// TIA Portal project "3M-9" (V16)

(* hardware
DEVICE "S7-1200 station_1"  S7-1200 Station
   slot 0: "Rack_0"  S7-1200 Rack  Rack  V1.0
   slot 1: "PLC_1"  CPU 1212C AC/DC/Rly  6ES7 212-1BE40-0XB0  V4.4
*)

// ===== PLC "PLC_1"  CPU 1212C AC/DC/Rly =====

VAR_GLOBAL   // PLC tag table "Default tag table"
   "START" AT %I0.0 : Bool;
   "STOP" AT %I0.1 : Bool;
   "MOTOR1" AT %Q0.0 : Bool;
   "MOTOR2" AT %Q0.1 : Bool;
   "MOTOR3" AT %Q0.2 : Bool;
   "X" AT %M0.0 : Bool;
   "Case 1" AT %M0.1 : Bool;
   "Case 2" AT %M0.2 : Bool;
   "Case 3" AT %M0.3 : Bool;
   "Y" AT %M0.4 : Bool;
   "tm1" AT %M0.5 : Bool;
   "tm2" AT %M0.6 : Bool;
   "TM3" AT %M0.7 : Bool;
   "SAVE Y" AT %M1.0 : Bool;
   "SAVE Z" AT %M1.1 : Bool;
END_VAR

// folder: System blocks/Program resources

DATA_BLOCK "timer1"   // DB1
{ S7_Optimized_Access := 'TRUE' }
AUTHOR : Simatic
FAMILY : IEC
NAME : IEC_TMR
VERSION : 1.0
// stored: InstanceOfName IEC_TIMER
"IEC_TIMER"
BEGIN
END_DATA_BLOCK

DATA_BLOCK "TIMER2"   // DB2
{ S7_Optimized_Access := 'TRUE' }
AUTHOR : Simatic
FAMILY : IEC
NAME : IEC_TMR
VERSION : 1.0
// stored: InstanceOfName IEC_TIMER
"IEC_TIMER"
BEGIN
END_DATA_BLOCK

DATA_BLOCK "TIMER3"   // DB3
{ S7_Optimized_Access := 'TRUE' }
AUTHOR : Simatic
FAMILY : IEC
NAME : IEC_TMR
VERSION : 1.0
// stored: InstanceOfName IEC_TIMER
"IEC_TIMER"
BEGIN
END_DATA_BLOCK

// folder: (top level)

ORGANIZATION_BLOCK "Main"   // OB1, LAD, ProgramCycle
TITLE = "Main Program Sweep (Cycle)"
{ S7_Optimized_Access := 'TRUE' }
VERSION : 0.1
   VAR_INPUT
      Initial_Call : Bool;   // Initial call of this OB
      Remanence : Bool;   // =True, if remanent data are available
   END_VAR
BEGIN

REGION Network 1
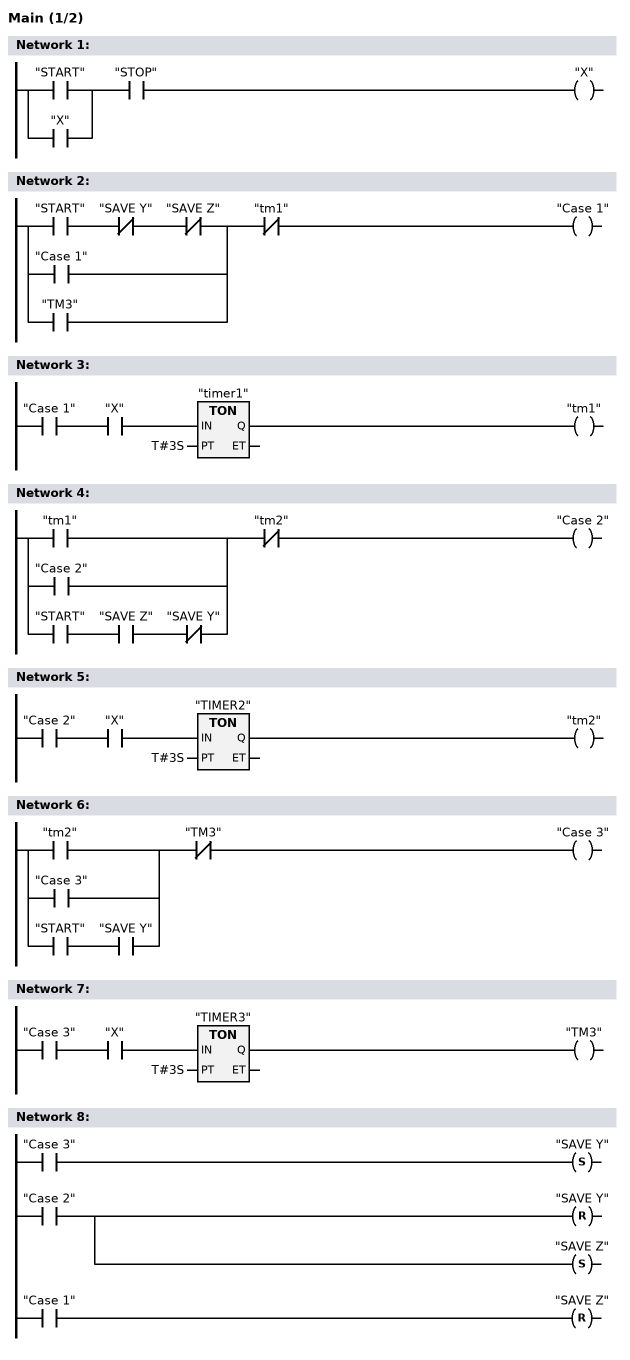
   RUNG wire#powerrail
      Contact( "START" )
      wire#w1
      Contact( "STOP" )
      Coil( "X" )
   END_RUNG
   RUNG wire#powerrail
      Contact( "X" )
   END_RUNG wire#w1
   // the same network as SCL:
   "X" := ("START" OR "X") AND "STOP";
END_REGION

REGION Network 2
   RUNG wire#powerrail
      Contact( "START" )
      I_Contact( "SAVE Y" )
      I_Contact( "SAVE Z" )
      wire#w1
      I_Contact( "tm1" )
      Coil( "Case 1" )
   END_RUNG
   RUNG wire#powerrail
      Contact( "Case 1" )
   END_RUNG wire#w1
   RUNG wire#powerrail
      Contact( "TM3" )
   END_RUNG wire#w1
   // the same network as SCL:
   "Case 1" := (("START" AND NOT "SAVE Y" AND NOT "SAVE Z") OR "Case 1" OR "TM3") AND NOT "tm1";
END_REGION

REGION Network 3
   "timer1".TON(IN := "Case 1" AND "X", PT := T#3S);
   "tm1" := "timer1".Q;
END_REGION

REGION Network 4
   RUNG wire#powerrail
      Contact( "tm1" )
      wire#w1
      I_Contact( "tm2" )
      Coil( "Case 2" )
   END_RUNG
   RUNG wire#powerrail
      Contact( "Case 2" )
   END_RUNG wire#w1
   RUNG wire#powerrail
      Contact( "START" )
      Contact( "SAVE Z" )
      I_Contact( "SAVE Y" )
   END_RUNG wire#w1
   // the same network as SCL:
   "Case 2" := ("tm1" OR "Case 2" OR ("START" AND "SAVE Z" AND NOT "SAVE Y")) AND NOT "tm2";
END_REGION

REGION Network 5
   "TIMER2".TON(IN := "Case 2" AND "X", PT := T#3S);
   "tm2" := "TIMER2".Q;
END_REGION

REGION Network 6
   RUNG wire#powerrail
      Contact( "tm2" )
      wire#w1
      I_Contact( "TM3" )
      Coil( "Case 3" )
   END_RUNG
   RUNG wire#powerrail
      Contact( "Case 3" )
   END_RUNG wire#w1
   RUNG wire#powerrail
      Contact( "START" )
      Contact( "SAVE Y" )
   END_RUNG wire#w1
   // the same network as SCL:
   "Case 3" := ("tm2" OR "Case 3" OR ("START" AND "SAVE Y")) AND NOT "TM3";
END_REGION

REGION Network 7
   "TIMER3".TON(IN := "Case 3" AND "X", PT := T#3S);
   "TM3" := "TIMER3".Q;
END_REGION

REGION Network 8
   RUNG wire#powerrail
      Contact( "Case 3" )
      S_Coil( "SAVE Y" )
   END_RUNG
   RUNG wire#powerrail
      Contact( "Case 2" )
      wire#w1
      R_Coil( "SAVE Y" )
   END_RUNG
   RUNG wire#w1
      S_Coil( "SAVE Z" )
   END_RUNG
   RUNG wire#powerrail
      Contact( "Case 1" )
      R_Coil( "SAVE Z" )
   END_RUNG
   // the same network as SCL:
   IF "Case 3" THEN "SAVE Y" := TRUE; END_IF;
   IF "Case 2" THEN
       "SAVE Y" := FALSE;
       "SAVE Z" := TRUE;
   END_IF;
   IF "Case 1" THEN "SAVE Z" := FALSE; END_IF;
END_REGION

REGION Network 9
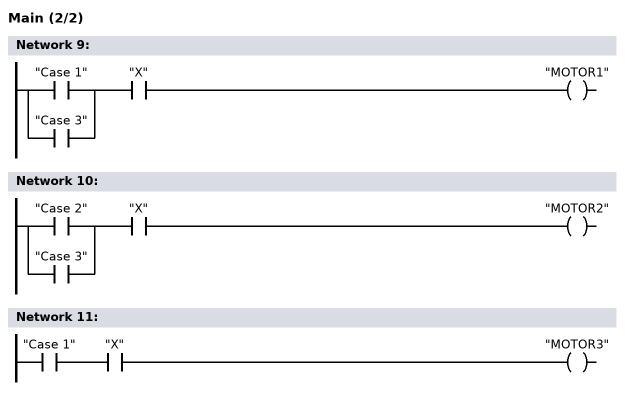
   RUNG wire#powerrail
      Contact( "Case 1" )
      wire#w1
      Contact( "X" )
      Coil( "MOTOR1" )
   END_RUNG
   RUNG wire#powerrail
      Contact( "Case 3" )
   END_RUNG wire#w1
   // the same network as SCL:
   "MOTOR1" := ("Case 1" OR "Case 3") AND "X";
END_REGION

REGION Network 10
   RUNG wire#powerrail
      Contact( "Case 2" )
      wire#w1
      Contact( "X" )
      Coil( "MOTOR2" )
   END_RUNG
   RUNG wire#powerrail
      Contact( "Case 3" )
   END_RUNG wire#w1
   // the same network as SCL:
   "MOTOR2" := ("Case 2" OR "Case 3") AND "X";
END_REGION

REGION Network 11
   RUNG wire#powerrail
      Contact( "Case 1" )
      Contact( "X" )
      Coil( "MOTOR3" )
   END_RUNG
   // the same network as SCL:
   "MOTOR3" := "Case 1" AND "X";
END_REGION
END_ORGANIZATION_BLOCK